FUNCTION_BLOCK DummyControl (* Basic Function Block Type *)
  (* Standard: 61499-2 *)
  (* Version 0.0, 6/17/2016, Andrei, nxtControl GmbH, Template *)
  PACKAGE Main;
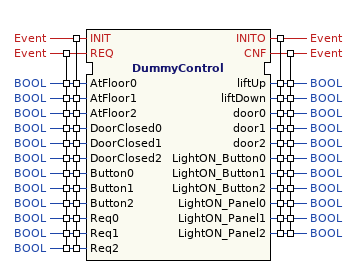
  EVENT_INPUT
    INIT WITH AtFloor0, AtFloor1, AtFloor2, DoorClosed0, DoorClosed1, DoorClosed2, Button0, Button1, Button2, Req0, Req1, Req2; (* Initialization Request *)
    REQ WITH AtFloor0, AtFloor1, AtFloor2, DoorClosed0, DoorClosed1, DoorClosed2, Button0, Button1, Button2, Req0, Req1, Req2; (* Normal Execution Request *)
  END_EVENT
  EVENT_OUTPUT
    INITO WITH liftUp, liftDown, door0, door1, door2, LightON_Button0, LightON_Button1, LightON_Button2, LightON_Panel0, LightON_Panel1, LightON_Panel2; (* Initialization Confirm *)
    CNF WITH liftUp, liftDown, door0, door1, door2, LightON_Button0, LightON_Button1, LightON_Button2, LightON_Panel0, LightON_Panel1, LightON_Panel2; (* Execution Confirmation *)
  END_EVENT
  VAR_INPUT
    AtFloor0 : BOOL; (* Input event qualifier *)
    AtFloor1 : BOOL;
    AtFloor2 : BOOL;
    DoorClosed0 : BOOL;
    DoorClosed1 : BOOL;
    DoorClosed2 : BOOL;
    Button0 : BOOL;
    Button1 : BOOL;
    Button2 : BOOL;
    Req0 : BOOL;
    Req1 : BOOL;
    Req2 : BOOL;
  END_VAR
  VAR_OUTPUT
    liftUp : BOOL;
    liftDown : BOOL; (* Output event qualifier *)
    door0 : BOOL;
    door1 : BOOL;
    door2 : BOOL;
    LightON_Button0 : BOOL;
    LightON_Button1 : BOOL;
    LightON_Button2 : BOOL;
    LightON_Panel0 : BOOL;
    LightON_Panel1 : BOOL;
    LightON_Panel2 : BOOL;
  END_VAR
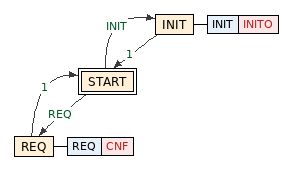
  EC_STATES
    START; (* Initial State *)
    INIT : INIT -> INITO; (* Initialization *)
    REQ : REQ -> CNF; (* Normal execution *)
  END_STATES
  EC_TRANSITIONS
    START TO INIT := INIT;
    INIT TO START := 1;
    START TO REQ := REQ;
    REQ TO START := 1;
  END_TRANSITIONS
  ALGORITHM INIT IN ST: (* Initialization algorithm *)
liftDown := TRUE;
  END_ALGORITHM
  ALGORITHM REQ IN ST: (* Normally executed algorithm *)
IF AtFloor0 THEN
	liftUp := TRUE;
	liftDown := FALSE;
END_IF;
IF AtFloor2 THEN
	liftDown := TRUE;
	liftUp := FALSE;
END_IF;

/*IF Button0 OR Req0 THEN
	door0 := TRUE;
ELSE
	door0 := FALSE;
END_IF;
IF Button1 OR Req1 THEN
	door1 := TRUE;
ELSE
	door1 := FALSE;
END_IF;
IF Button2 OR Req2 THEN
	door2 := TRUE;
ELSE
	door2 := FALSE;
END_IF;*/
door0 := Button0 OR Req0;
door1 := Button1 OR Req1;
door2 := Button2 OR Req2;

LightON_Button0 := Button0;
LightON_Button1 := Button1;
LightON_Button2 := Button2;

LightON_Panel0 := Req0;
LightON_Panel1 := Req1;
LightON_Panel2 := Req2;
  END_ALGORITHM
END_FUNCTION_BLOCK
